SUBAPPLICATION Uebung_090a1 (* Beispiel für F_MUX_2 *)
  (* Standard: 61499-2; Description: Copyright (c) 2023 Meisterschulen am Ostbahnhof This program and the accompanying materials are made available under the terms of the Eclipse Public License 2.0 which is available at https://www.eclipse.org/legal/epl-2.0/ SPDX-License-Identifier: EPL-2.0 *)
  (* Version 1.0, 2023-10-23, Franz Höpfinger, Meisterschulen am Ostbahnhof *)
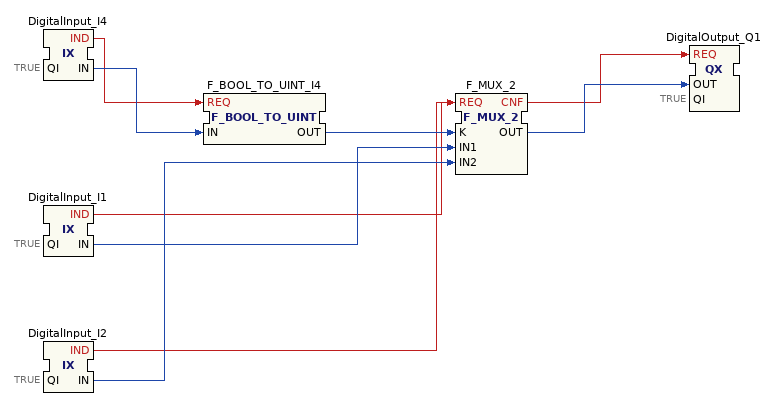
  FBS
    F_MUX_2 : F_MUX_2;
    DigitalInput_I4 : IX(QI := TRUE);
    F_BOOL_TO_UINT_I4 : F_BOOL_TO_UINT;
    DigitalOutput_Q1 : QX(QI := TRUE);
    DigitalInput_I1 : IX(QI := TRUE);
    DigitalInput_I2 : IX(QI := TRUE);
  END_FBS
  EVENT_CONNECTIONS
    DigitalInput_I4.IND TO F_BOOL_TO_UINT_I4.REQ;
    F_MUX_2.CNF TO DigitalOutput_Q1.REQ;
    DigitalInput_I1.IND TO F_MUX_2.REQ;
    DigitalInput_I2.IND TO F_MUX_2.REQ;
  END_CONNECTIONS
  DATA_CONNECTIONS
    DigitalInput_I4.IN TO F_BOOL_TO_UINT_I4.IN;
    F_BOOL_TO_UINT_I4.OUT TO F_MUX_2.K;
    F_MUX_2.OUT TO DigitalOutput_Q1.OUT;
    DigitalInput_I1.IN TO F_MUX_2.IN1;
    DigitalInput_I2.IN TO F_MUX_2.IN2;
  END_CONNECTIONS
END_SUBAPPLICATION
